FUNCTION_BLOCK CHIP_REMOVAL_ON_OFF (* Activates chip removal *)
  (* Standard: 61499-2 *)
  (* Version 1.0, 09-01-12, Guilherme Jarentchuk, Universidade do Estado de Santa Catarina *)
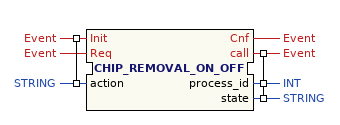
  EVENT_INPUT
    Init WITH action; (* Initialize execution *)
    Req; (* Request to finish *)
  END_EVENT
  EVENT_OUTPUT
    Cnf; (* Confirm execution *)
    call WITH state, process_id; (* Call execution device *)
  END_EVENT
  VAR_INPUT
    action : STRING; (* Can be only "on" or "off" *)
  END_VAR
  VAR_OUTPUT
    process_id : INT;
    state : STRING;
  END_VAR
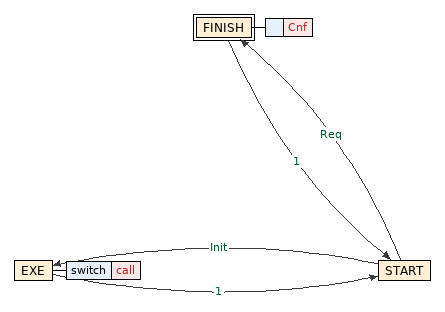
  EC_STATES
    FINISH : -> Cnf;
    START;
    EXE : switch -> call;
  END_STATES
  EC_TRANSITIONS
    FINISH TO START := 1;
    START TO EXE := Init;
    START TO FINISH := Req;
    EXE TO START := 1;
  END_TRANSITIONS
  ALGORITHM switch IN Lua:
 if( action == "on" ) or ( action == "true" ) then
    state = "on"
elseif( action == "off" ) or ( action == "false" )  then
    state = "off"
end
process_id = -4
  END_ALGORITHM
END_FUNCTION_BLOCK
